PROGRAM P_Safety
VAR
END_VAR

GVL_Safety.bErrAck := GVL_IO.arrDIs[8];

END_PROGRAM

(* stored: Version 1.1.0.1
   POU P_Safety: Id {3af665d7-6873-4846-8277-a5c5c53e4398}, SpecialFunc None *)
